# EPICS autosave request: soft_iocs/toaster/iocBoot/ioctoaster/ao.req
$(P)$(D)$(R).VAL
$(P)$(D)$(R).DRVH
$(P)$(D)$(R).DRVL
$(P)$(D)$(R).DESC
$(P)$(D)$(R).EGU
$(P)$(D)$(R).PREC
